Fanuc TP program (LS listing): MAKRO050.LS

/PROG  MAKRO050
/ATTR
OWNER		= MNEDITOR;
COMMENT		= "Merkerbildung";
PROG_SIZE	= 2780;
CREATE		= DATE 20-12-22  TIME 17:29:08;
MODIFIED	= DATE 23-12-11  TIME 08:28:16;
FILE_NAME	= ;
VERSION		= 0;
LINE_COUNT	= 104;
MEMORY_SIZE	= 3152;
PROTECT		= READ_WRITE;
TCD:  STACK_SIZE	= 0,
      TASK_PRIORITY	= 50,
      TIME_SLICE	= 0,
      BUSY_LAMP_OFF	= 0,
      ABORT_REQUEST	= 0,
      PAUSE_REQUEST	= 0;
DEFAULT_GROUP	= *,*,*,*,*;
CONTROL_CODE	= 00000000 00000000;
/MN
   1:  !Merker-Init ;
   2:  !Roboter mit Greifer. ;
   3:  !Dual Sta. EZ ohne KW. ;
   4:  ! ;
   5:  !Abfrage Bauteilkontrollen ;
   6:  M[1]=((DI[605] AND DI[607]) OR DI[15]) ;
   7:  M[2]=(!DI[605] AND !DI[607]) ;
   8:  ! ;
   9:  !Abfrage Spanngruppen ;
  10:  M[31]=(!DI[579] AND DI[580] AND !DI[581] AND DI[582]) ;
  11:  M[32]=(DI[579] AND !DI[580] AND DI[581] AND !DI[582]) ;
  12:  M[33]=(DI[583] AND !DI[584] AND DI[585] AND !DI[586] AND DI[587] AND !DI[588] AND DI[589] AND !DI[590]) ;
  13:  M[34]=(!DI[583] AND DI[584] AND !DI[585] AND DI[586] AND !DI[587] AND DI[588] AND !DI[589] AND DI[590]) ;
  14:  M[35]=(OFF) ;
  15:  M[36]=(OFF) ;
  16:  M[37]=(OFF) ;
  17:  M[38]=(OFF) ;
  18:  M[39]=(OFF) ;
  19:  M[40]=(OFF) ;
  20:  M[41]=(OFF) ;
  21:  M[42]=(OFF) ;
  22:  M[43]=(OFF) ;
  23:  M[44]=(OFF) ;
  24:  M[45]=(OFF) ;
  25:  M[46]=(OFF) ;
  26:  M[47]=(OFF) ;
  27:  M[48]=(OFF) ;
  28:  M[49]=(OFF) ;
  29:  M[50]=(OFF) ;
  30:  M[51]=(OFF) ;
  31:  M[52]=(OFF) ;
  32:  M[53]=(OFF) ;
  33:  M[54]=(OFF) ;
  34:  M[55]=(OFF) ;
  35:  M[56]=(OFF) ;
  36:  M[57]=(OFF) ;
  37:  M[58]=(OFF) ;
  38:  M[59]=(OFF) ;
  39:  M[60]=(OFF) ;
  40:  M[61]=(OFF) ;
  41:  M[62]=(OFF) ;
  42:  M[63]=(OFF) ;
  43:  M[64]=(OFF) ;
  44:  M[65]=(OFF) ;
  45:  M[66]=(OFF) ;
  46:  M[67]=(OFF) ;
  47:  M[68]=(OFF) ;
  48:  ! ;
  49:  !Maschinelle Sicherheiten ;
  50:  !mit Niederdruck ueberwachung ;
  51:  M[30]=(DI[14] AND DI[24] AND DI[516] AND DI[524]) ;
  52:  ! ;
  53:  !Widerstandspunktschweissen ;
  54:  !Sicherheiten EZ1/SP1 ;
  55:  M[95]=(DI[705] AND !DI[706] AND DI[713] AND DI[714] AND ((!DI[715] AND DI[719]) OR DO[715]) AND !DI[773] AND !DI[779] AND DO[716]) ;
  56:  !Grundstellung KS1 ;
  57:  M[96]=(DI[842] AND !DI[844] AND !DI[843] AND DI[845] AND !DO[715] AND (F[321] OR (DO[875] AND F[148]) OR (DO[1035] AND F[184]))) ;
  58:  !Flankenausw.der Fraeserumd.KF1 ;
  59:  M[97]=((DI[718] AND DO[718] OR F[312]) AND DI[834] AND DO[834] AND !F[72] AND !F[73] AND (F[90] OR F[92])) ;
  60:  !Sicherheiten EZ2/SP2 ;
  61:  M[102]=(DI[865] AND !DI[866] AND DI[873] AND DI[874] AND ((!DI[875] AND DI[879]) OR DO[875]) AND !DI[933] AND !DI[939] AND DO[876]) ;
  62:  !Grundstellung KS2 ;
  63:  M[103]=(DI[1002] AND !DI[1004] AND !DI[1003] AND DI[1005] AND !DO[875] AND (F[321] OR (DO[715] AND F[92]) OR (DO[1035] AND F[148]))) ;
  64:  !Flankenausw.der Fraeserumd.KF2 ;
  65:  M[104]=((DI[878] AND DO[878] OR F[312]) AND DI[994] AND DO[994] AND F[148]) ;
  66:  ! ;
  67:  !EZ1/SP1/SZ1 Umdrehungen Startfr ;
  68:  R[2]=4    ;
  69:  !Umdrehungen Startfraesen Teil 2 ;
  70:  R[3]=4    ;
  71:  !Umdrehungen Nomalfraesen ;
  72:  R[4]=3    ;
  73:  !EZ1/SP1/SZ2 Umdrehungen Startfr ;
  74:  R[5]=8    ;
  75:  !Umdrehungen Startfraesen Teil 2 ;
  76:  R[6]=8    ;
  77:  !Umdrehungen Nomalfraesen ;
  78:  R[7]=8    ;
  79:  !min. Oeffnung stat. EZ/SP ;
  80:  !beim Fraesen ;
  81:  R[60]=600    ;
  82:  ! ;
  83:  !;Ausgleichswert EZ1/SP1 ;
  84:  R[197]=113    ;
  85:  !;Ausgleichswert EZ2/SP2 ;
  86:  R[198]=114    ;
  87:  !Kappenverschl. Verhaeltnis ;
  88:  !feste EK in % (Stat-EZ1) ;
  89:  R[411]=65    ;
  90:  !Kappenverschl. Verhaeltnis ;
  91:  !feste EK in % (Stat-EZ2) ;
  92:  R[412]=65    ;
  93:   ;
  94:  !Kappenkompenstion bei ;
  95:  !stationaerer EZ1/SP1 ;
  96:  CALL MOTN004    ;
  97:  !Kappenkompenstion bei ;
  98:  !stationaerer EZ2/SP2 ;
  99:  CALL MOTN005    ;
 100:  ! ;
 101:  !Aufruf Makro57 ;
 102:  CALL MAKRO057    ;
 103:  !Docking ;
 104:  CALL MAKRO058    ;
/POS
/END
